INTERFACE I_Motor

METHOD Start : BOOL
VAR_INPUT
END_VAR
END_METHOD

METHOD Stop : BOOL
VAR_INPUT
END_VAR
END_METHOD

END_INTERFACE

(* stored: Version 1.1.0.1, ProductVersion 3.1.4024.16
   Itf I_Motor: Id {412aa1d1-0f4f-4e11-9ff7-12ead4c3e809}
   Method Start: Id {0d873179-86d2-4b69-96eb-64e1e76c0c42}
   Method Stop: Id {1297f19c-c551-4d94-a0ed-9cb132401529} *)
